(* PLC project Cell Example , CTH FIX1 1.0, author CTH SS2 *)
(* stored: companyURL www.chalmers.se, creationDateTime 2008-03-19T20:31:26, version 1.0, modificationDateTime 2008-04-21T11:16:17, organization SS2, language en-US *)

TYPE BinaryPositions : ();
END_TYPE

FUNCTION_BLOCK RAC
  VAR_INPUT
    IN1 : BOOL := FALSE;
  END_VAR
  VAR_OUTPUT
    OUT : BOOL := FALSE;
  END_VAR
  VAR_INPUT
    IN2 : BOOL := FALSE;
  END_VAR
  VAR
    Var3 : BOOL := FALSE;
    Var4 : BOOL := FALSE;
  END_VAR
  VAR_INPUT
    IN5 : BOOL := FALSE;
    IN6 : BOOL := TRUE;
  END_VAR
  VAR
    Var7 : BOOL := TRUE;
  END_VAR
  VAR  (* added by the conversion: wires and edge detectors of the diagram *)
    R_TRIG1 : R_TRIG;
  END_VAR

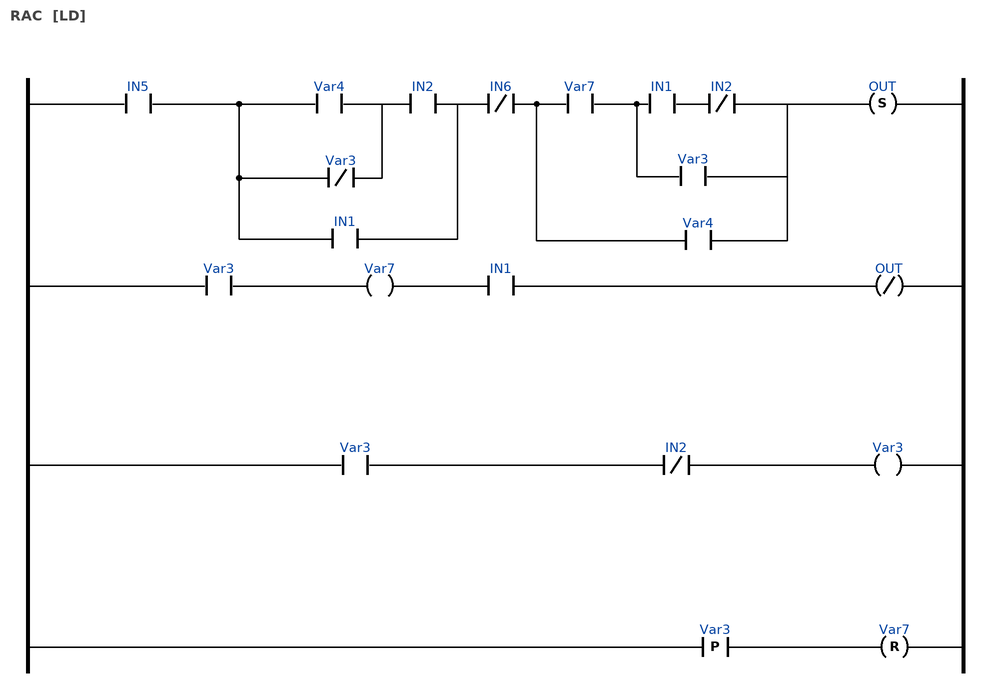
(* LD diagram, written out as Structured Text *)
IF IN5 AND ((NOT Var3 OR Var4) AND IN2 OR IN1) AND NOT IN6 AND (Var7 AND IN1 AND NOT IN2 OR Var7 AND Var3 OR Var4) THEN OUT := TRUE; END_IF;
Var7 := Var3;
OUT := NOT (Var3 AND IN1);
Var3 := Var3 AND NOT IN2;
R_TRIG1(CLK := Var3);
IF R_TRIG1.Q THEN Var7 := FALSE; END_IF;
END_FUNCTION_BLOCK

CONFIGURATION ExampleCell
END_CONFIGURATION
